(* IEC 61131-3 sources: HappyLearnCodesys/content/softmotion/CNC16_G31, 2 files *)

(* ---- Main.st ---- *)
PROGRAM Main
VAR_OUTPUT
    setStart: SMC_SetInterpreterStartPosition;
END_VAR
VAR
	pwX: MC_Power;
	pwY: MC_Power;
    ipo : SMC_Interpolator;
	capX: SMC_ControlAxisByPos;
	capY: SMC_ControlAxisByPos;
    trafo : SMC_TRAFO_Gantry2;
	trafoF: SMC_TRAFOF_Gantry2;
END_VAR

(* ---- Path.st ---- *)
PROGRAM Path
VAR_OUTPUT
    poqDataOut : POINTER TO SMC_OUTQUEUE;
END_VAR
VAR
    read : SMC_ReadNCFile2 := (sFileName:= 'Application/gcode.cnc');
    inter : SMC_NCInterpreter;
    cv : SMC_CheckVelocities;

    bufIpo : ARRAY[0..99] OF SMC_GEOINFO;
END_VAR

read(bExecute:= TRUE);

inter(
    sentences:= read.sentences,
    bExecute:= read.bExecute,
    nSizeOutQueue:= SIZEOF(bufIpo),
    pbyBufferOutQueue:= ADR(bufIpo),
	piStartPosition:= Main.setStart.StartPos);

cv(bExecute:= read.bExecute,
   poqDataIn:= inter.poqDataOut);

poqDataOut := cv.poqDataOut;
